// TIA Portal V16 export
// export: Created 2020-03-17T19:45:03.5424607Z, ExportSetting None, DisplayName Totally Integrated Automation Portal, DisplayVersion V16, DisplayName TIA Portal Version Control Interface, DisplayVersion V16, DisplayName TIA Portal Openness, DisplayVersion V16, DisplayName STEP 7 Professional, DisplayVersion V16, DisplayName STEP 7 Safety, DisplayVersion V16, DisplayName WinCC Advanced, DisplayVersion V16
FUNCTION_BLOCK "FB_R134a_GRAPH"   // FB1308, GRAPH
// stored: GraphVersion 2.0, SetENOAutomatically false
   // inherited from GRAPH_BASE
   VAR_INPUT
      OFF_SQ { ExternalAccessible := 'False'; ExternalVisible := 'False'; ExternalWritable := 'False'} : Bool := false;   // Kette ausschalten / Turn sequence off
      INIT_SQ { ExternalAccessible := 'False'; ExternalVisible := 'False'; ExternalWritable := 'False'} : Bool := false;   // Kette in Initialzustand versetzen / Set sequence to initial state
      ACK_EF { ExternalAccessible := 'False'; ExternalVisible := 'False'; ExternalWritable := 'False'} : Bool := false;   // Alle Fehler und Störungen quittieren / Acknowledge all errors and faults
      S_PREV { ExternalAccessible := 'False'; ExternalVisible := 'False'; ExternalWritable := 'False'} : Bool := false;   // Vorherigen Schritt am Parameter S_NO ausgeben / Output previous step in parameter S_NO
      S_NEXT { ExternalAccessible := 'False'; ExternalVisible := 'False'; ExternalWritable := 'False'} : Bool := false;   // Nächsten Schritt am Parameter S_NO anzeigen / Indicate next step in parameter S_NO
      SW_AUTO { ExternalAccessible := 'False'; ExternalVisible := 'False'; ExternalWritable := 'False'} : Bool := false;   // Automatischer Betrieb / Automatic mode
      SW_TAP { ExternalAccessible := 'False'; ExternalVisible := 'False'; ExternalWritable := 'False'} : Bool := false;   // Halbautomatisch/Weiterschalten mit Transition / Semiautomatic/switch with transition
      SW_TOP { ExternalAccessible := 'False'; ExternalVisible := 'False'; ExternalWritable := 'False'} : Bool := false;   // Halbautomatisch/Ignoriere Transition / Semiautomatic/ignore transition
      SW_MAN { ExternalAccessible := 'False'; ExternalVisible := 'False'; ExternalWritable := 'False'} : Bool := false;   // Handbetrieb / Manual mode
      S_SEL { ExternalAccessible := 'False'; ExternalVisible := 'False'; ExternalWritable := 'False'} : Int := 0;   // Schritt auswählen, der an S_NO ausgegeben werden soll / Select step to be output to S_NO
      S_ON { ExternalAccessible := 'False'; ExternalVisible := 'False'; ExternalWritable := 'False'} : Bool := false;   // Schritt aktivieren, der an Parameter S_NO anliegt / Activate step indicated in S_NO
      S_OFF { ExternalAccessible := 'False'; ExternalVisible := 'False'; ExternalWritable := 'False'} : Bool := false;   // Schritt deaktivieren, der an Parameter S_NO anliegt / Deactivate step indicated S_NO
      T_PUSH { ExternalAccessible := 'False'; ExternalVisible := 'False'; ExternalWritable := 'False'} : Bool := false;   // Schaltfreigabe für Transition im halbautomatischen Betrieb / Enable transition to switch in semi automatic mode
   END_VAR
   VAR_OUTPUT
      S_NO { ExternalAccessible := 'False'; ExternalVisible := 'False'; ExternalWritable := 'False'} : Int := 0;   // Schrittnummer / Step number
      S_MORE { ExternalAccessible := 'False'; ExternalVisible := 'False'; ExternalWritable := 'False'} : Bool := false;   // Weitere Schritte sind vorhanden und können in S_NO angezeigt werden. / More steps are available and can be shown in S_NO
      S_ACTIVE { ExternalAccessible := 'False'; ExternalVisible := 'False'; ExternalWritable := 'False'} : Bool := false;   // Schritt, der an Parameter S_NO angezeigt wird, ist aktiv / Step indicated in S_NO is active
      ERR_FLT { ExternalAccessible := 'False'; ExternalVisible := 'False'; ExternalWritable := 'False'} : Bool := false;   // Sammelfehler Interlock oder Supervision / Interlock or supervision group error
      AUTO_ON { ExternalAccessible := 'False'; ExternalVisible := 'False'; ExternalWritable := 'False'} : Bool := false;   // Automatischer Betrieb eingeschaltet / Automatic mode is active
      TAP_ON { ExternalAccessible := 'False'; ExternalVisible := 'False'; ExternalWritable := 'False'} : Bool := false;   // Halbautomatischer Betrieb/Schritt mit Transition eingeschaltet / Semiautomatic mode/step with transition enabled
      TOP_ON { ExternalAccessible := 'False'; ExternalVisible := 'False'; ExternalWritable := 'False'} : Bool := false;   // Halbautomatischer Betrieb/Ignoriere Transition eingeschaltet / Semiautomatic mode/ignore transition enabled
      MAN_ON { ExternalAccessible := 'False'; ExternalVisible := 'False'; ExternalWritable := 'False'} : Bool := false;   // Handbetrieb eingeschaltet / Manual mode is active
   END_VAR
BEGIN
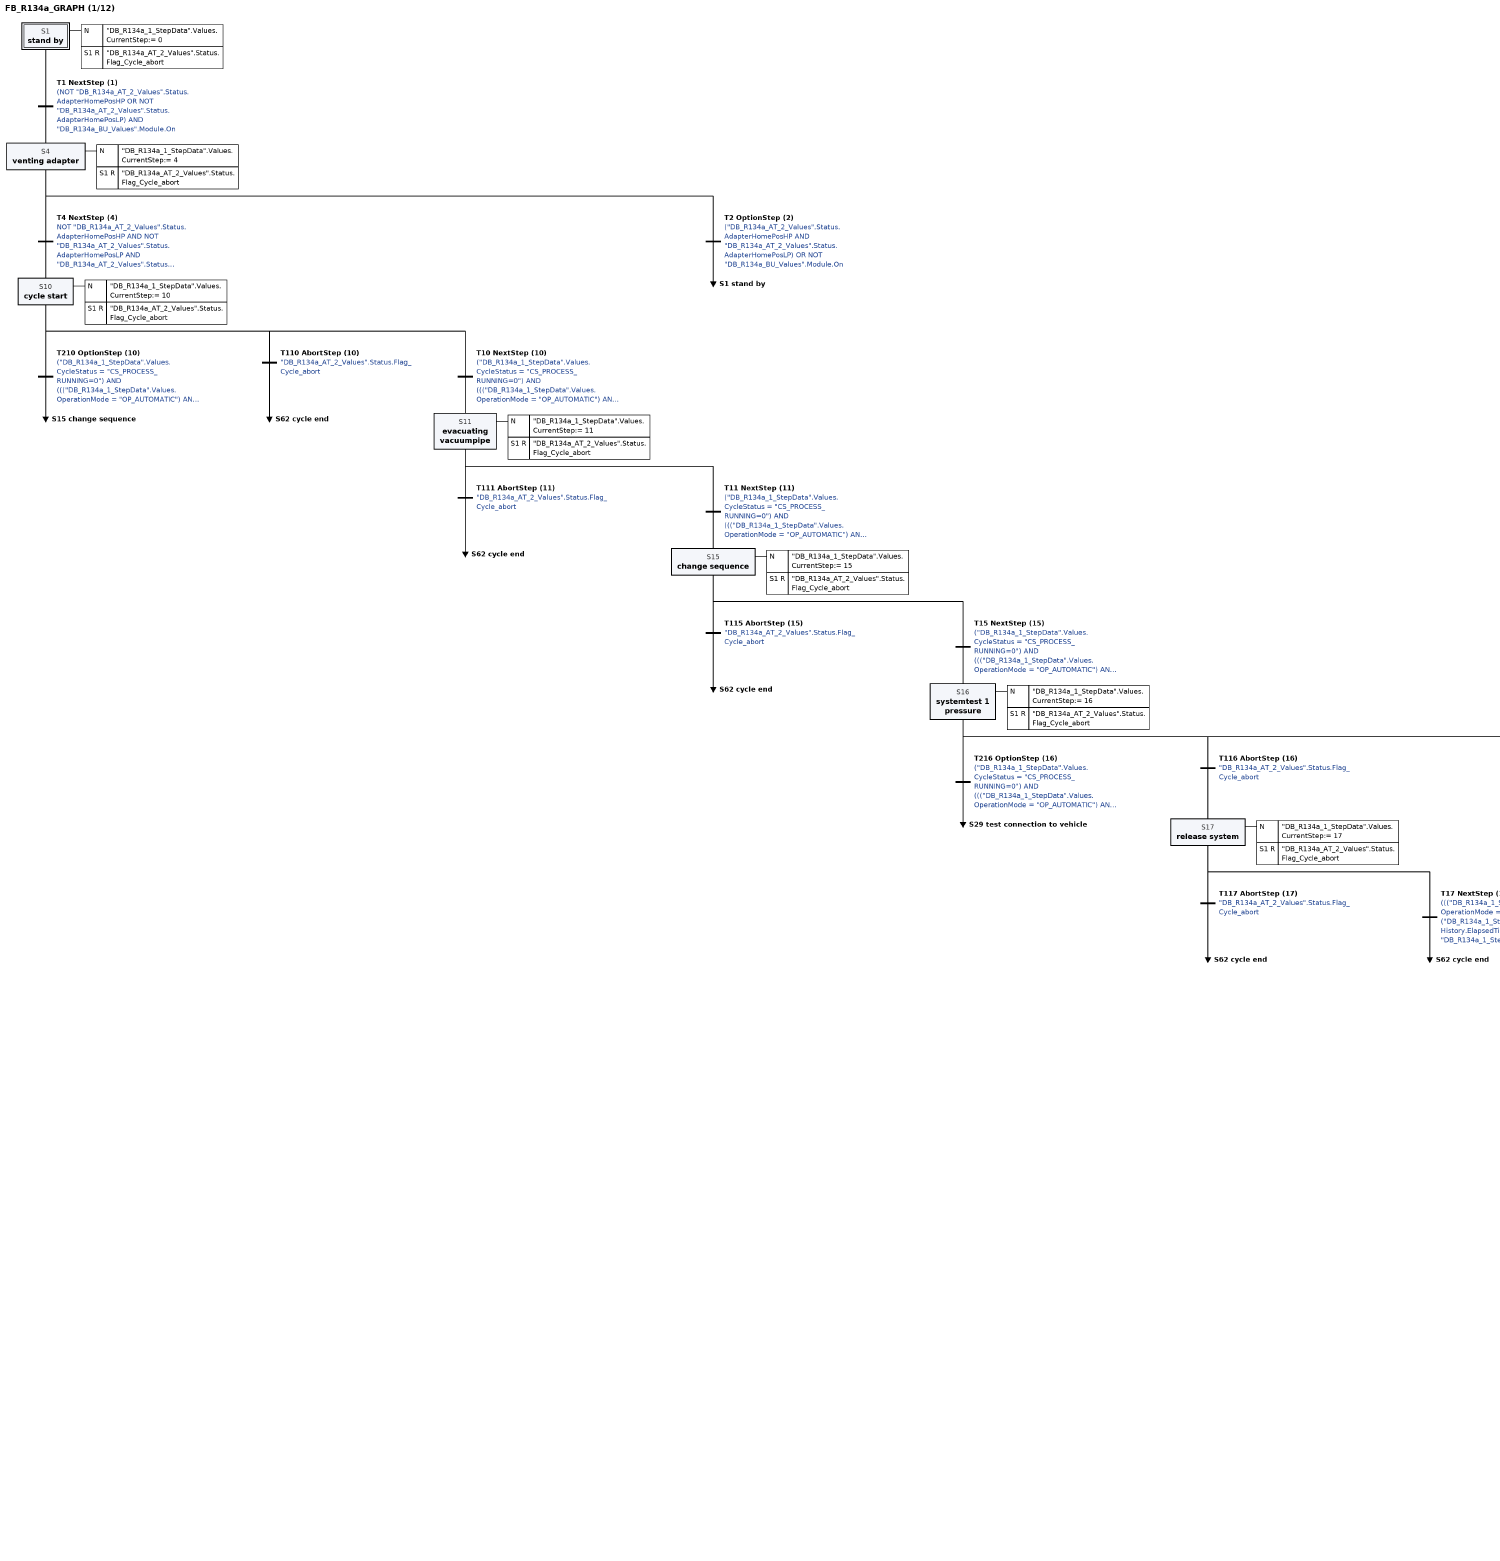
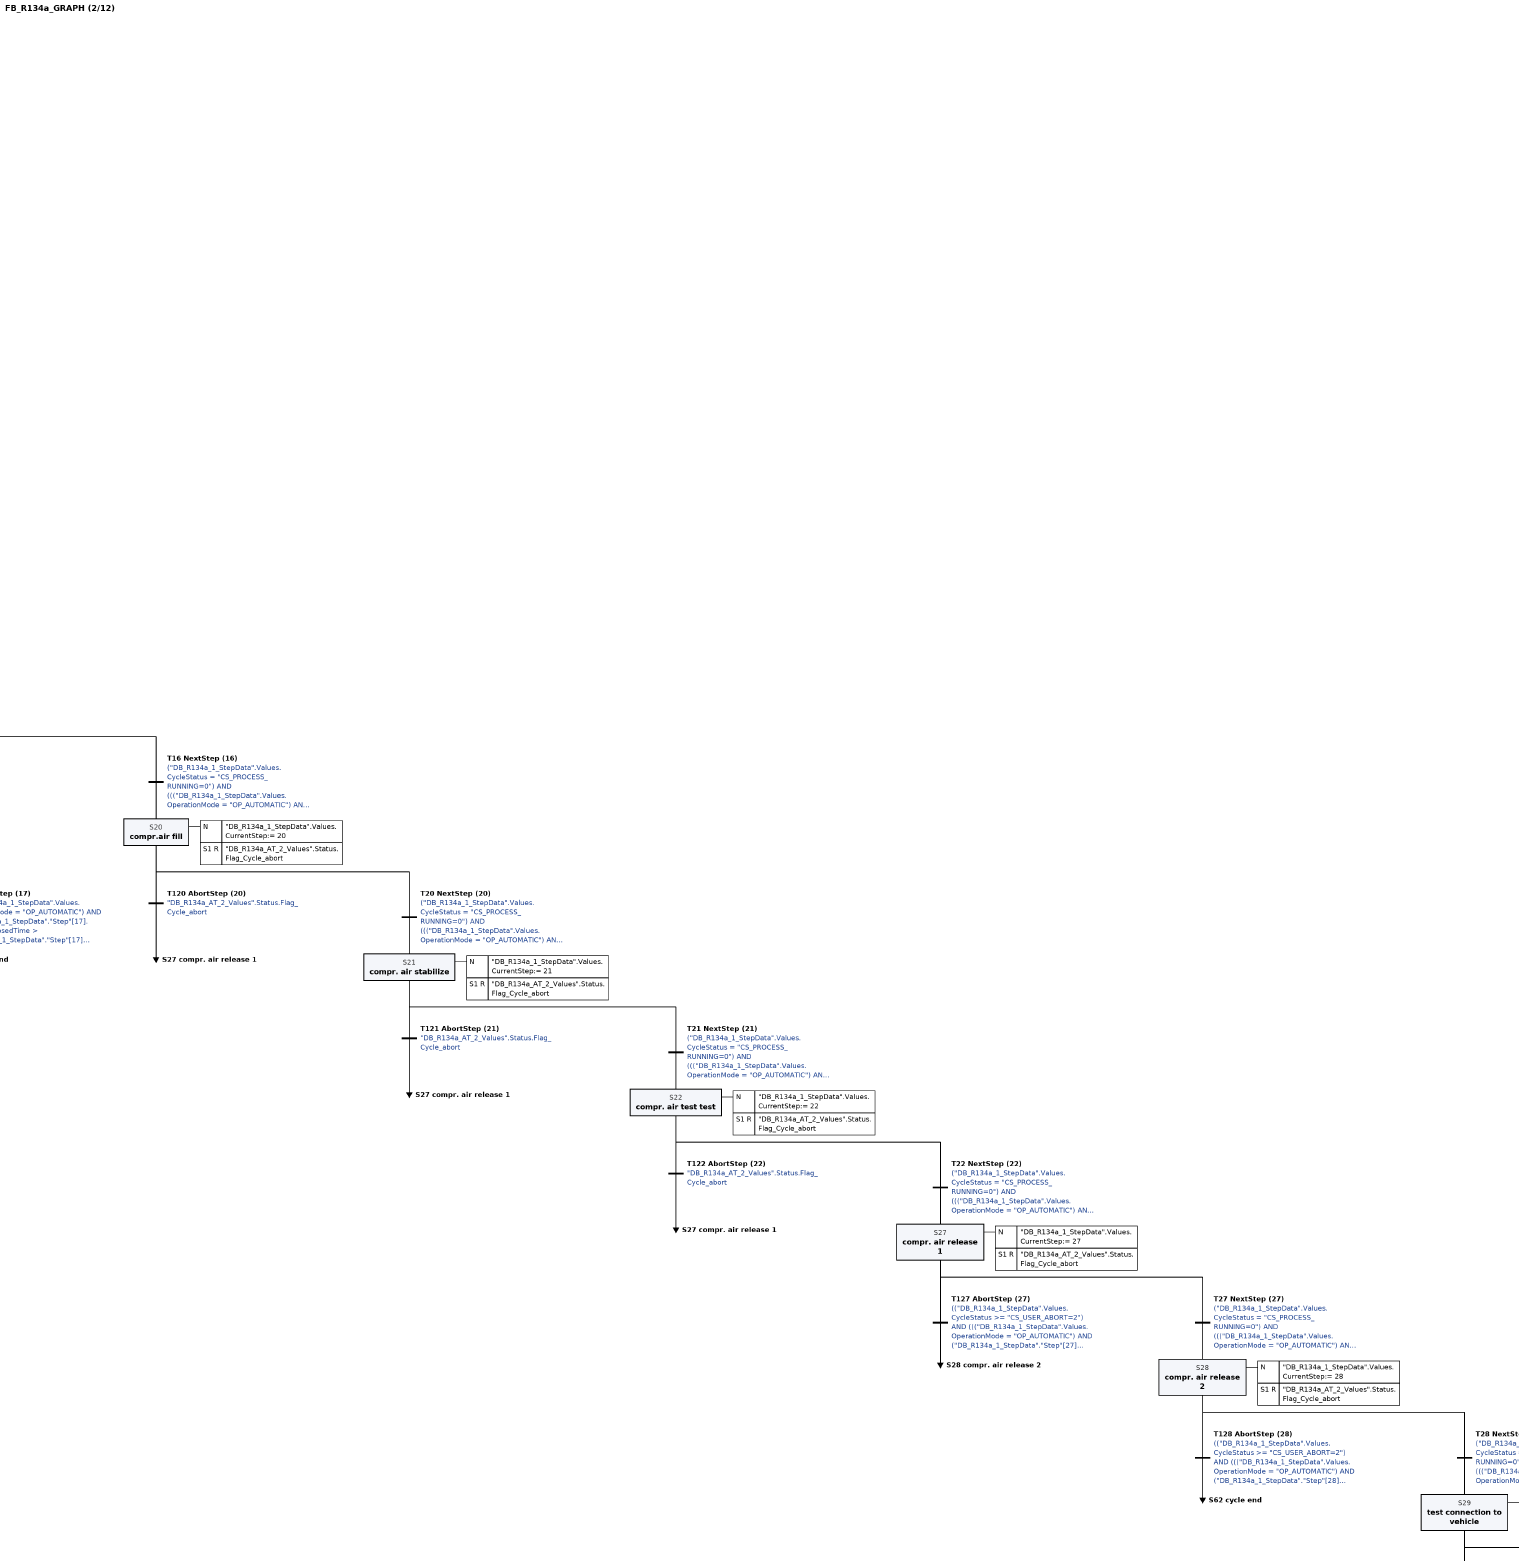
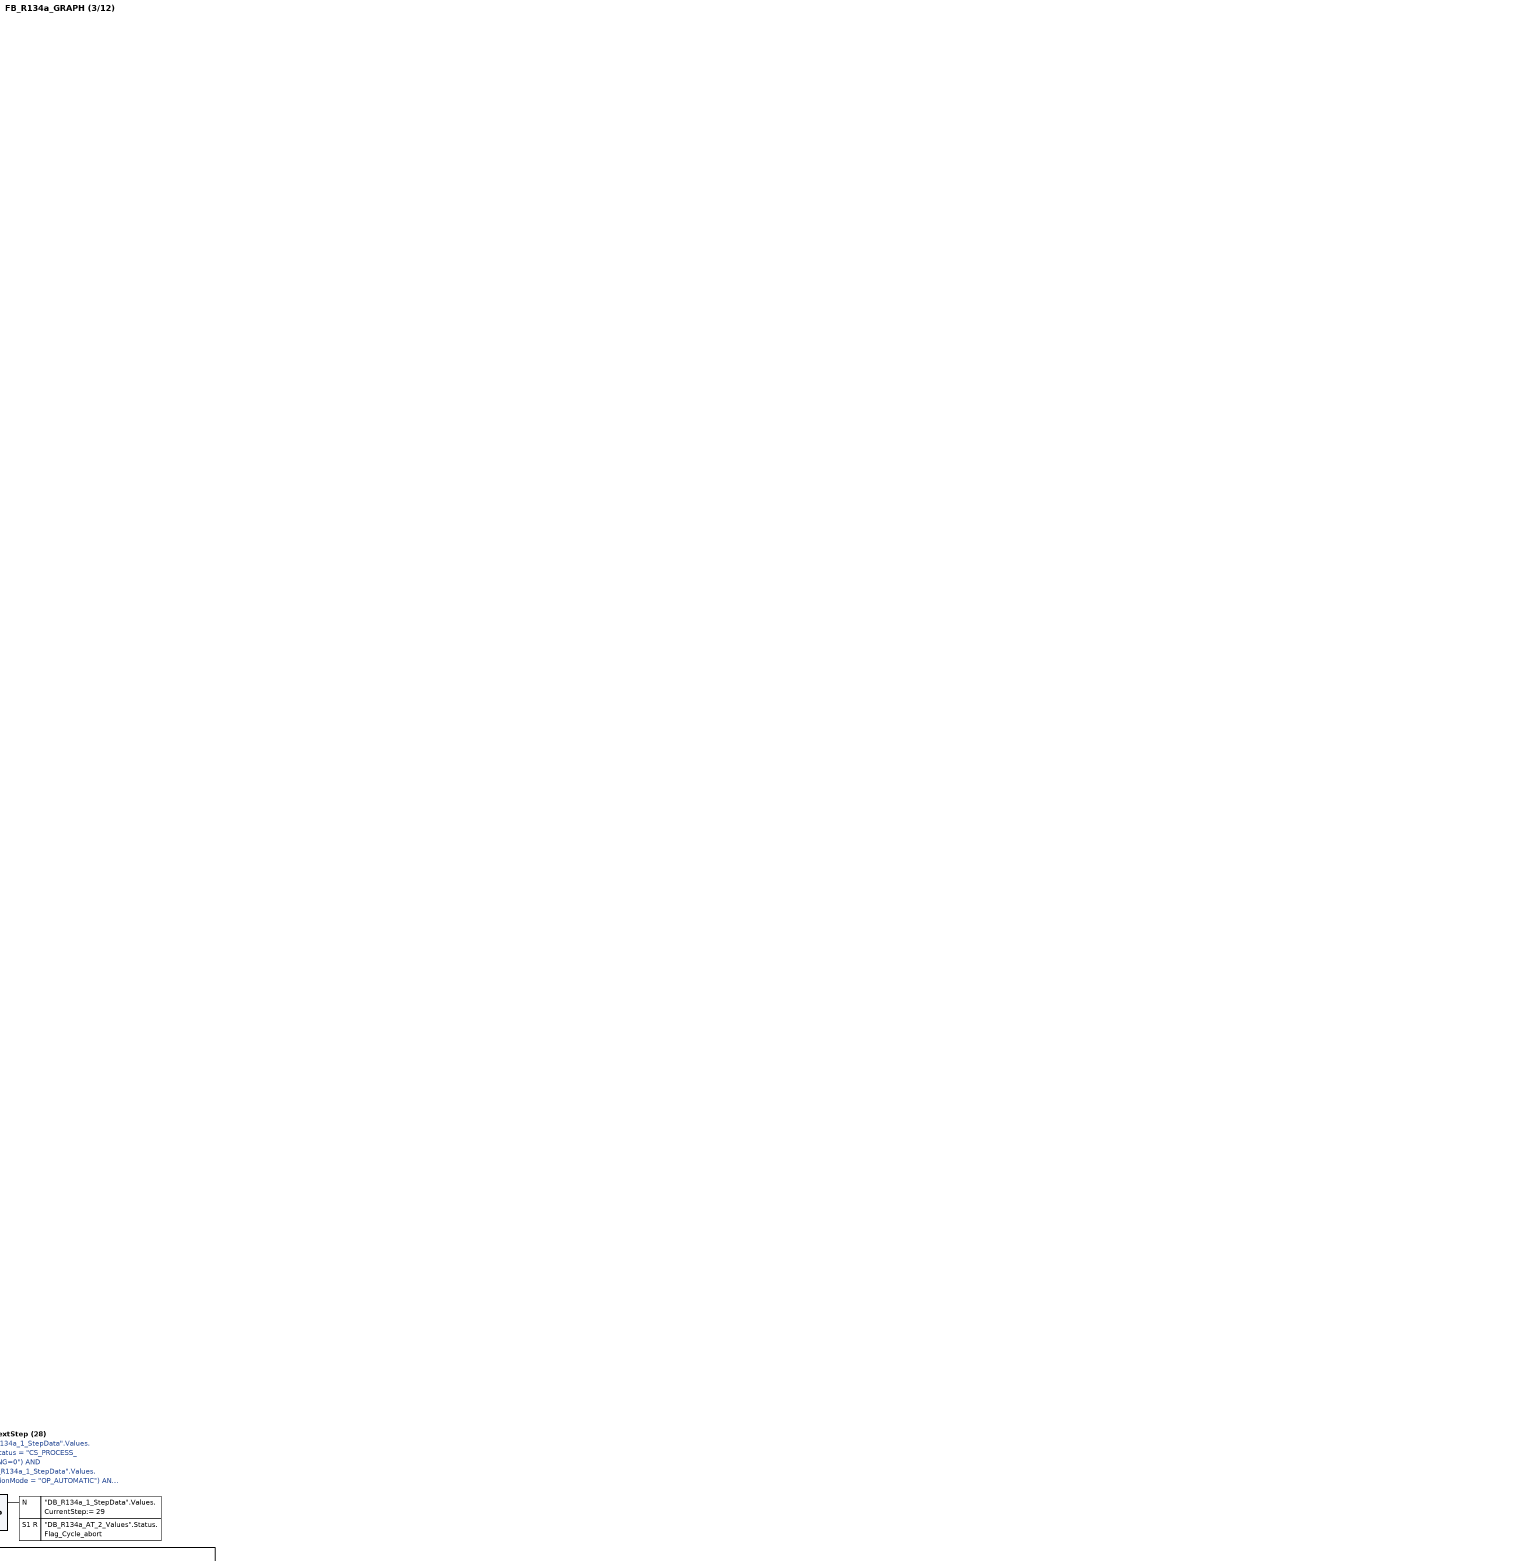
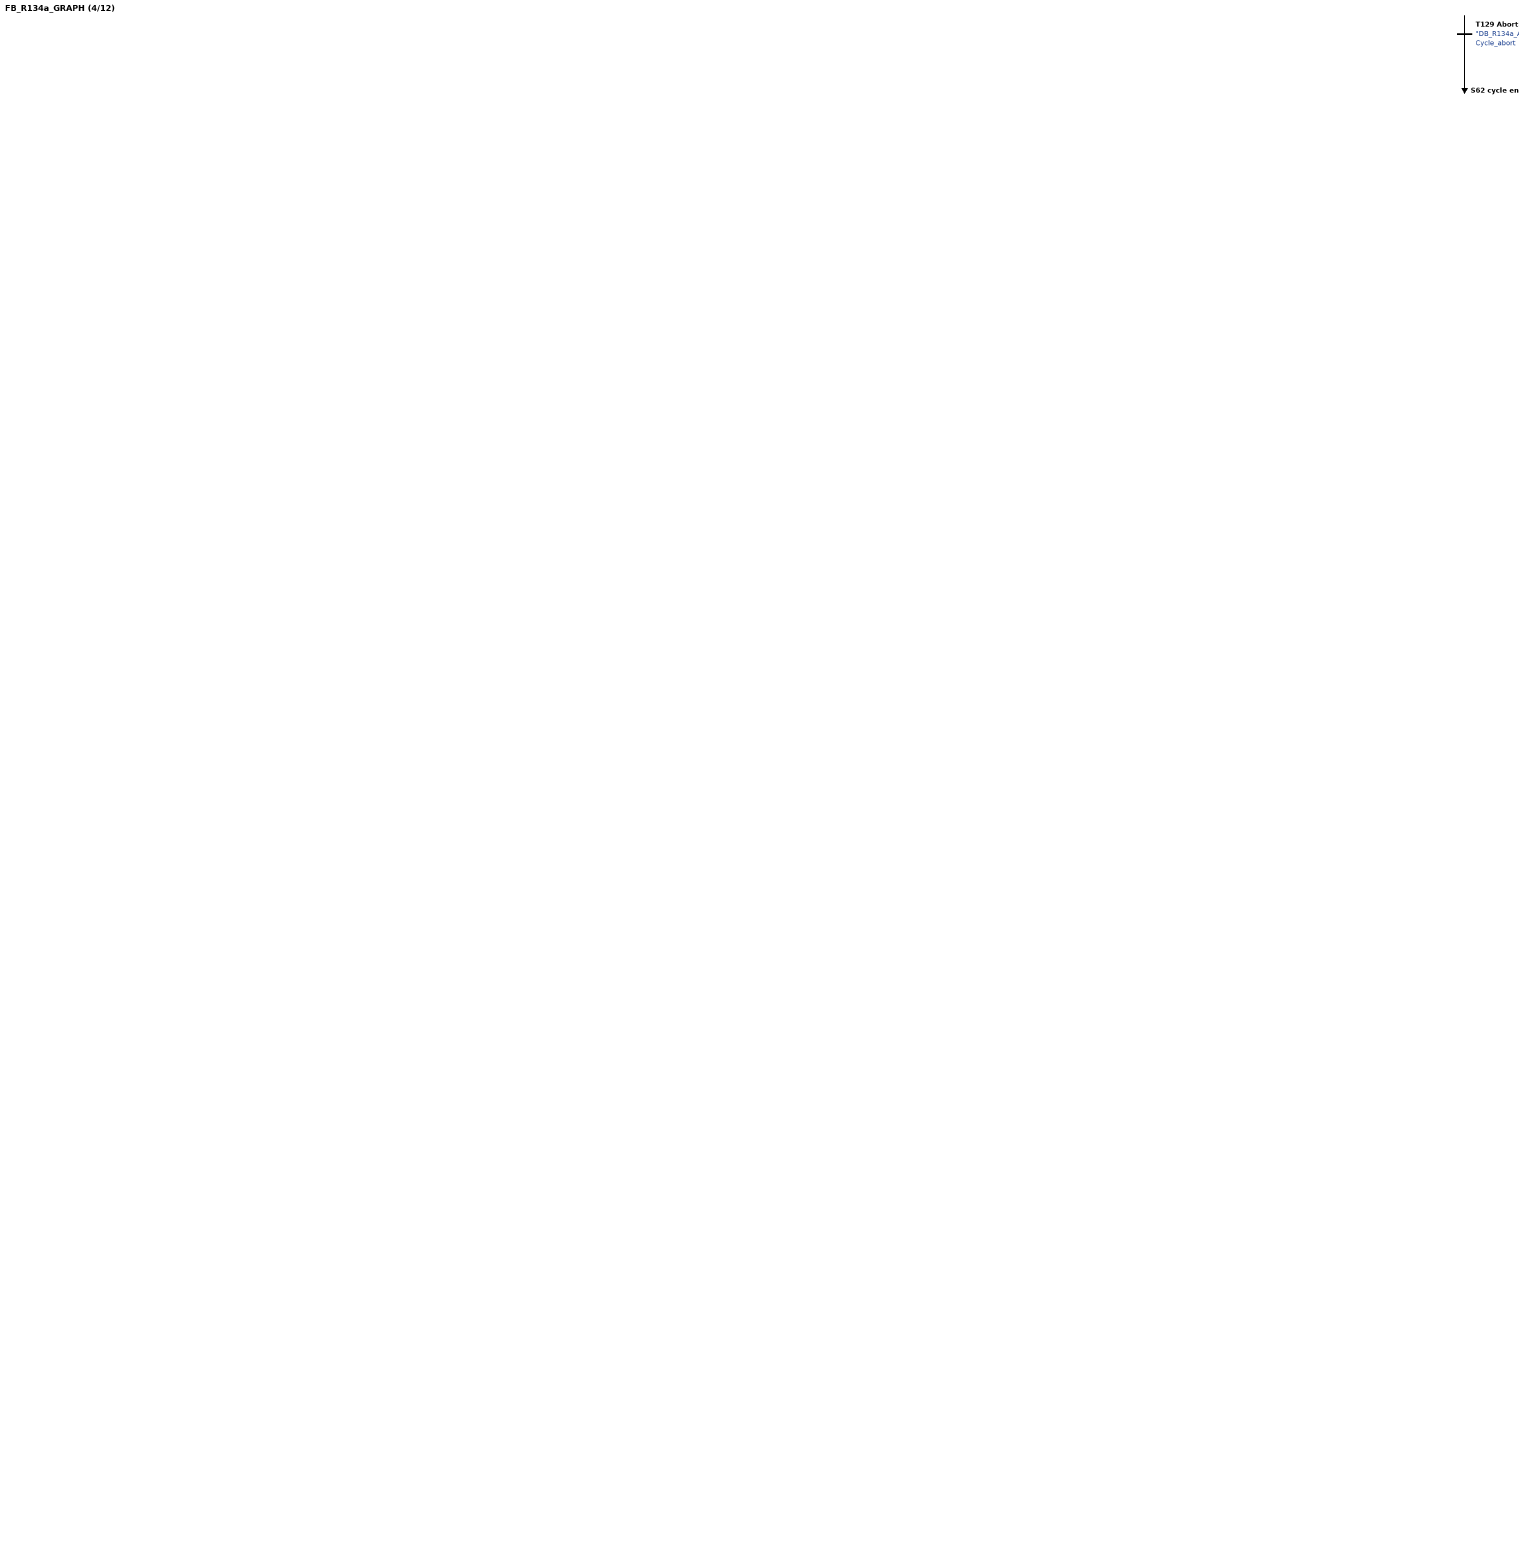
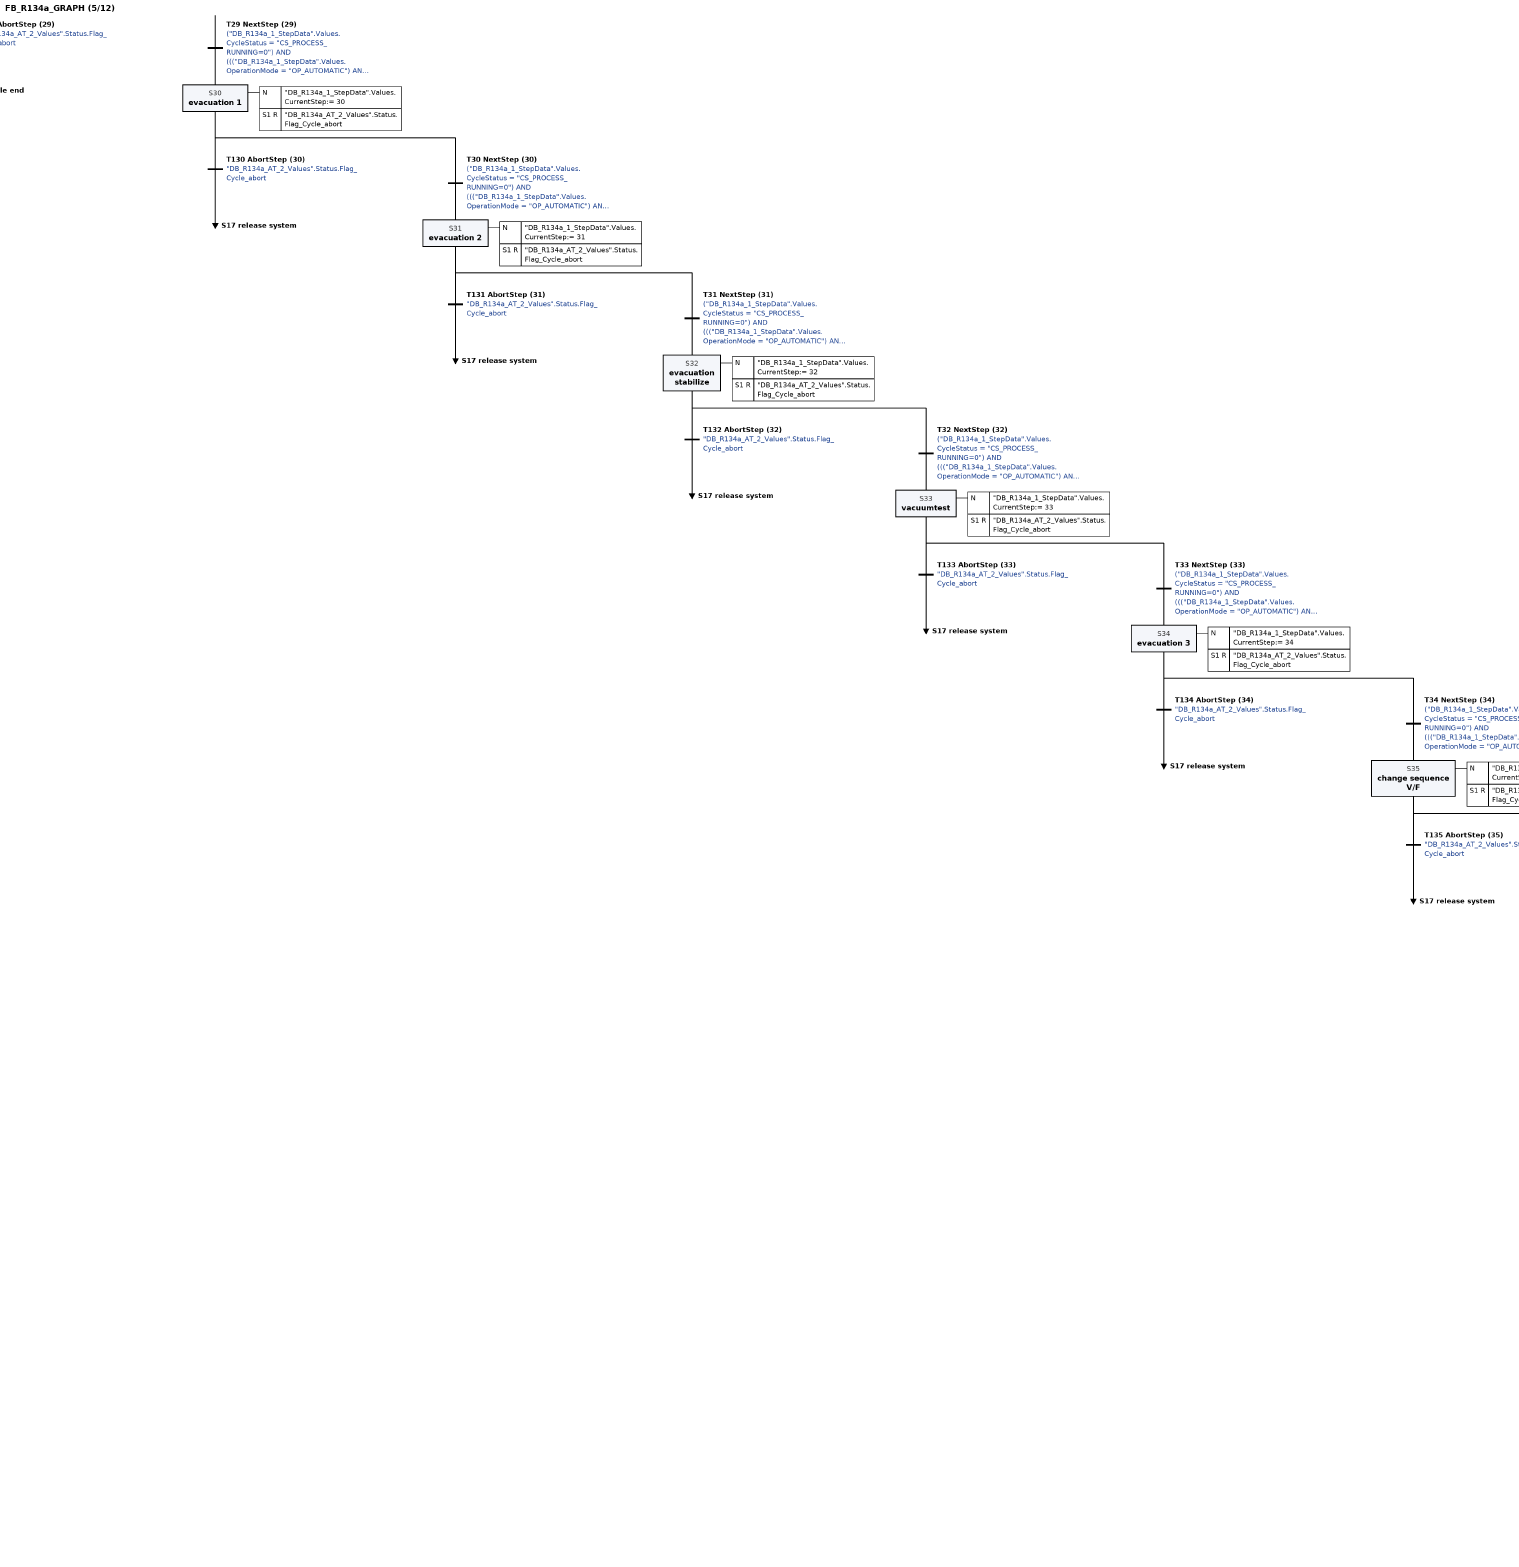
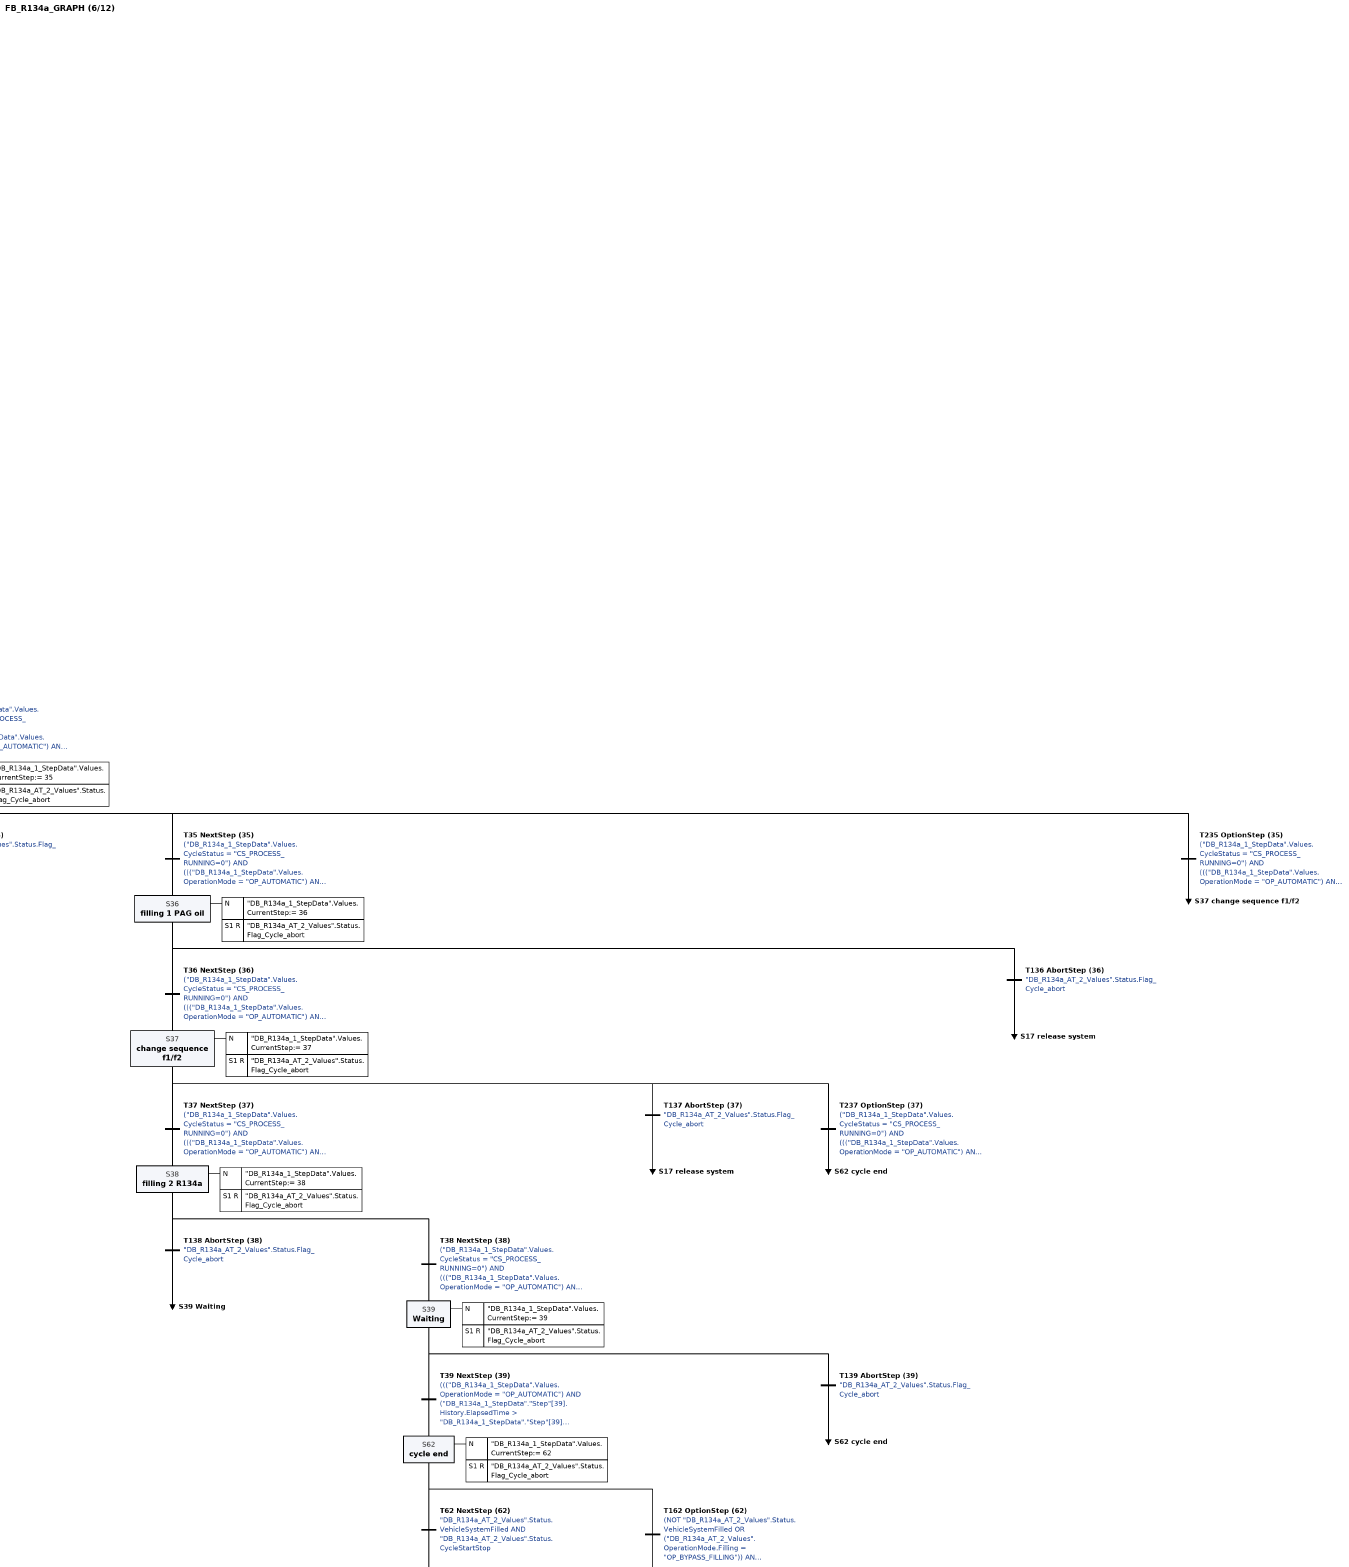
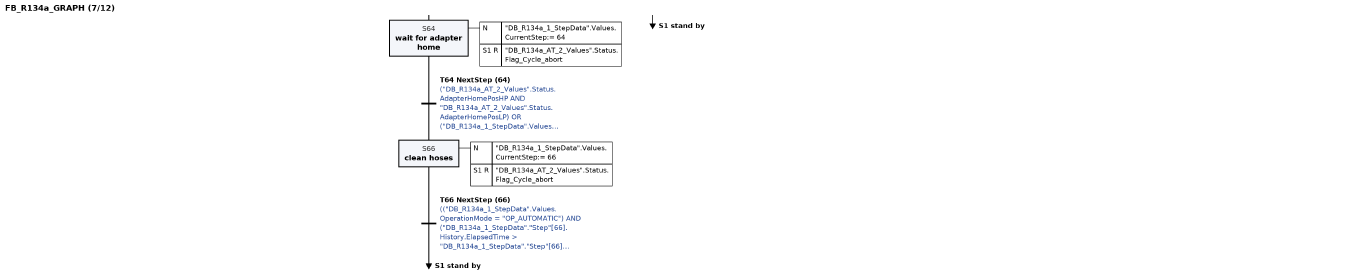
   // sequencer 1
   STEP "release system":   // S17, max time T#10S, warning time T#7S
              N    "DB_R134a_1_StepData".Values.CurrentStep:= 17
          S1  R    "DB_R134a_AT_2_Values".Status.Flag_Cycle_abort
   END_STEP
   TRANSITION "AbortStep (17)" FROM "release system" TO "cycle end"   // T117, jump
      := "DB_R134a_AT_2_Values".Status.Flag_Cycle_abort;
   END_TRANSITION
   TRANSITION "NextStep (17)" FROM "release system" TO "cycle end"   // T17, jump
      := ((("DB_R134a_1_StepData".Values.OperationMode = "OP_AUTOMATIC") AND ("DB_R134a_1_StepData"."Step"[17].History.ElapsedTime > "DB_R134a_1_StepData"."Step"[17].WaitingTime)) OR ("DB_R134a_1_StepData".Values.SingleStep AND ("DB_R134a_1_StepData".Values.OperationMode = "OP_SingleStep"))) AND NOT "DB_R134a_AT_2_Values".Status.Flag_Cycle_abort;
   END_TRANSITION
   STEP "clean hoses":   // S66, max time T#10S, warning time T#7S
              N    "DB_R134a_1_StepData".Values.CurrentStep:= 66
          S1  R    "DB_R134a_AT_2_Values".Status.Flag_Cycle_abort
   END_STEP
   TRANSITION "NextStep (66)" FROM "clean hoses" TO "stand by"   // T66, jump
      := (("DB_R134a_1_StepData".Values.OperationMode = "OP_AUTOMATIC") AND ("DB_R134a_1_StepData"."Step"[66].History.ElapsedTime > "DB_R134a_1_StepData"."Step"[66].WaitingTime)) OR ("DB_R134a_1_StepData".Values.SingleStep AND ("DB_R134a_1_StepData".Values.OperationMode = "OP_SingleStep"));
   END_TRANSITION
   STEP "wait for adapter home":   // S64, max time T#10S, warning time T#7S
              N    "DB_R134a_1_StepData".Values.CurrentStep:= 64
          S1  R    "DB_R134a_AT_2_Values".Status.Flag_Cycle_abort
   END_STEP
   TRANSITION "NextStep (64)" FROM "wait for adapter home" TO "clean hoses"   // T64
      := ("DB_R134a_AT_2_Values".Status.AdapterHomePosHP AND "DB_R134a_AT_2_Values".Status.AdapterHomePosLP) OR ("DB_R134a_1_StepData".Values.SingleStep AND ("DB_R134a_1_StepData".Values.OperationMode = "OP_SingleStep"));
   END_TRANSITION
   STEP "cycle end":   // S62, max time T#10S, warning time T#7S
              N    "DB_R134a_1_StepData".Values.CurrentStep:= 62
          S1  R    "DB_R134a_AT_2_Values".Status.Flag_Cycle_abort
   END_STEP
   TRANSITION "NextStep (62)" FROM "cycle end" TO "wait for adapter home"   // T62
      := "DB_R134a_AT_2_Values".Status.VehicleSystemFilled AND "DB_R134a_AT_2_Values".Status.CycleStartStop;
   END_TRANSITION
   TRANSITION "OptionStep (62)" FROM "cycle end" TO "stand by"   // T162, jump
      := (NOT "DB_R134a_AT_2_Values".Status.VehicleSystemFilled OR ("DB_R134a_AT_2_Values".OperationMode.Filling = "OP_BYPASS_FILLING")) AND "DB_R134a_AT_2_Values".Status.CycleStartStop;
   END_TRANSITION
   STEP Waiting:   // S39, max time T#10S, warning time T#7S
              N    "DB_R134a_1_StepData".Values.CurrentStep:= 39
          S1  R    "DB_R134a_AT_2_Values".Status.Flag_Cycle_abort
   END_STEP
   TRANSITION "NextStep (39)" FROM Waiting TO "cycle end"   // T39
      := ((("DB_R134a_1_StepData".Values.OperationMode = "OP_AUTOMATIC") AND ("DB_R134a_1_StepData"."Step"[39].History.ElapsedTime > "DB_R134a_1_StepData"."Step"[39].WaitingTime)) OR ("DB_R134a_1_StepData".Values.SingleStep AND ("DB_R134a_1_StepData".Values.OperationMode = "OP_SingleStep"))) AND NOT "DB_R134a_AT_2_Values".Status.Flag_Cycle_abort;
   END_TRANSITION
   TRANSITION "AbortStep (39)" FROM Waiting TO "cycle end"   // T139, jump
      := "DB_R134a_AT_2_Values".Status.Flag_Cycle_abort;
   END_TRANSITION
   STEP "filling 2 R134a":   // S38, max time T#10S, warning time T#7S
      supervision V := ("DB_R134a_1_StepData".Values.OperationMode <> "OP_SingleStep") AND (#"filling 2 R134a".U > "DB_R134a_1_StepData"."Step"[38].MonitoringTime) AND ("DB_R134a_1_StepData".Values.CycleStatus = "CS_PROCESS_RUNNING=0");
              N    "DB_R134a_1_StepData".Values.CurrentStep:= 38
          S1  R    "DB_R134a_AT_2_Values".Status.Flag_Cycle_abort
   END_STEP
   TRANSITION "AbortStep (38)" FROM "filling 2 R134a" TO Waiting   // T138, jump
      := "DB_R134a_AT_2_Values".Status.Flag_Cycle_abort;
   END_TRANSITION
   TRANSITION "NextStep (38)" FROM "filling 2 R134a" TO Waiting   // T38
      := ("DB_R134a_1_StepData".Values.CycleStatus = "CS_PROCESS_RUNNING=0") AND ((("DB_R134a_1_StepData".Values.OperationMode = "OP_AUTOMATIC") AND ("DB_R134a_1_StepData"."Step"[38].History.ElapsedTime > "DB_R134a_1_StepData"."Step"[38].WaitingTime) AND "DB_R134a_BU_Values".Flowmeter.Output.VolumeDone) OR ("DB_R134a_1_StepData".Values.SingleStep AND ("DB_R134a_1_StepData".Values.OperationMode = "OP_SingleStep"))) AND NOT "DB_R134a_AT_2_Values".Status.Flag_Cycle_abort;
   END_TRANSITION
   STEP "change sequence V/F":   // S35, max time T#10S, warning time T#7S
              N    "DB_R134a_1_StepData".Values.CurrentStep:= 35
          S1  R    "DB_R134a_AT_2_Values".Status.Flag_Cycle_abort
   END_STEP
   TRANSITION "AbortStep (35)" FROM "change sequence V/F" TO "release system"   // T135, jump
      := "DB_R134a_AT_2_Values".Status.Flag_Cycle_abort;
   END_TRANSITION
   TRANSITION "NextStep (35)" FROM "change sequence V/F" TO "filling 1 PAG oil"   // T35
      := ("DB_R134a_1_StepData".Values.CycleStatus = "CS_PROCESS_RUNNING=0") AND ((("DB_R134a_1_StepData".Values.OperationMode = "OP_AUTOMATIC") AND ("DB_R134a_1_StepData"."Step"[35].History.ElapsedTime > "DB_R134a_1_StepData"."Step"[35].WaitingTime)) OR ("DB_R134a_1_StepData".Values.SingleStep AND ("DB_R134a_1_StepData".Values.OperationMode = "OP_SingleStep"))) AND ("DB_R134a_AT_2_Values".OperationMode.FillingPAG = "OP_WITH_PAG") AND NOT "DB_R134a_AT_2_Values".Status.Flag_Cycle_abort;
   END_TRANSITION
   TRANSITION "OptionStep (35)" FROM "change sequence V/F" TO "change sequence f1/f2"   // T235, jump
      := ("DB_R134a_1_StepData".Values.CycleStatus = "CS_PROCESS_RUNNING=0") AND ((("DB_R134a_1_StepData".Values.OperationMode = "OP_AUTOMATIC") AND ("DB_R134a_1_StepData"."Step"[35].History.ElapsedTime > "DB_R134a_1_StepData"."Step"[35].WaitingTime)) OR ("DB_R134a_1_StepData".Values.SingleStep AND ("DB_R134a_1_StepData".Values.OperationMode = "OP_SingleStep"))) AND ("DB_R134a_AT_2_Values".OperationMode.FillingPAG = "OP_BYPASS_FILLING_PAG") AND NOT "DB_R134a_AT_2_Values".Status.Flag_Cycle_abort;
   END_TRANSITION
   STEP "evacuation 3":   // S34, max time T#10S, warning time T#7S
      supervision V := ("DB_R134a_1_StepData".Values.OperationMode <> "OP_SingleStep") AND (#"evacuation 3".U > "DB_R134a_1_StepData"."Step"[34].MonitoringTime) AND ("DB_R134a_1_StepData".Values.CycleStatus = "CS_PROCESS_RUNNING=0");
              N    "DB_R134a_1_StepData".Values.CurrentStep:= 34
          S1  R    "DB_R134a_AT_2_Values".Status.Flag_Cycle_abort
   END_STEP
   TRANSITION "AbortStep (34)" FROM "evacuation 3" TO "release system"   // T134, jump
      := "DB_R134a_AT_2_Values".Status.Flag_Cycle_abort;
   END_TRANSITION
   TRANSITION "NextStep (34)" FROM "evacuation 3" TO "change sequence V/F"   // T34
      := ("DB_R134a_1_StepData".Values.CycleStatus = "CS_PROCESS_RUNNING=0") AND ((("DB_R134a_1_StepData".Values.OperationMode = "OP_AUTOMATIC") AND ("DB_R134a_1_StepData"."Step"[34].History.ElapsedTime > "DB_R134a_1_StepData"."Step"[34].WaitingTime) AND ("DB_R134a_1_StepData"."Step"[34].History.Values[1] <= "DB_R134a_1_StepData"."Step"[34].Setpoint[1])) OR ("DB_R134a_1_StepData".Values.SingleStep AND ("DB_R134a_1_StepData".Values.OperationMode = "OP_SingleStep"))) AND NOT "DB_R134a_AT_2_Values".Status.Flag_Cycle_abort;
   END_TRANSITION
   STEP vacuumtest:   // S33, max time T#10S, warning time T#7S
      supervision V := ("DB_R134a_1_StepData".Values.OperationMode <> "OP_SingleStep") AND (#vacuumtest.U > "DB_R134a_1_StepData"."Step"[33].MonitoringTime) AND ("DB_R134a_1_StepData".Values.CycleStatus = "CS_PROCESS_RUNNING=0");
              N    "DB_R134a_1_StepData".Values.CurrentStep:= 33
          S1  R    "DB_R134a_AT_2_Values".Status.Flag_Cycle_abort
   END_STEP
   TRANSITION "AbortStep (33)" FROM vacuumtest TO "release system"   // T133, jump
      := "DB_R134a_AT_2_Values".Status.Flag_Cycle_abort;
   END_TRANSITION
   TRANSITION "NextStep (33)" FROM vacuumtest TO "evacuation 3"   // T33
      := ("DB_R134a_1_StepData".Values.CycleStatus = "CS_PROCESS_RUNNING=0") AND ((("DB_R134a_1_StepData".Values.OperationMode = "OP_AUTOMATIC") AND ("DB_R134a_1_StepData"."Step"[33].History.ElapsedTime > "DB_R134a_1_StepData"."Step"[33].WaitingTime) AND ("DB_R134a_1_StepData"."Step"[33].History.Values[1] <= "DB_R134a_1_StepData"."Step"[33].Setpoint[1]) AND ("DB_R134a_1_StepData"."Step"[33].History.Values[2] <= "DB_R134a_1_StepData"."Step"[33].Setpoint[2])) OR ("DB_R134a_1_StepData".Values.SingleStep AND ("DB_R134a_1_StepData".Values.OperationMode = "OP_SingleStep"))) AND NOT "DB_R134a_AT_2_Values".Status.Flag_Cycle_abort;
   END_TRANSITION
   STEP "evacuation stabilize":   // S32, max time T#10S, warning time T#7S
              N    "DB_R134a_1_StepData".Values.CurrentStep:= 32
          S1  R    "DB_R134a_AT_2_Values".Status.Flag_Cycle_abort
   END_STEP
   TRANSITION "AbortStep (32)" FROM "evacuation stabilize" TO "release system"   // T132, jump
      := "DB_R134a_AT_2_Values".Status.Flag_Cycle_abort;
   END_TRANSITION
   TRANSITION "NextStep (32)" FROM "evacuation stabilize" TO vacuumtest   // T32
      := ("DB_R134a_1_StepData".Values.CycleStatus = "CS_PROCESS_RUNNING=0") AND ((("DB_R134a_1_StepData".Values.OperationMode = "OP_AUTOMATIC") AND ("DB_R134a_1_StepData"."Step"[32].History.ElapsedTime > "DB_R134a_1_StepData"."Step"[32].WaitingTime)) OR ("DB_R134a_1_StepData".Values.SingleStep AND ("DB_R134a_1_StepData".Values.OperationMode = "OP_SingleStep"))) AND NOT "DB_R134a_AT_2_Values".Status.Flag_Cycle_abort;
   END_TRANSITION
   STEP "evacuation 2":   // S31, max time T#10S, warning time T#7S
      supervision V := ("DB_R134a_1_StepData".Values.OperationMode <> "OP_SingleStep") AND (#"evacuation 2".U > "DB_R134a_1_StepData"."Step"[31].MonitoringTime) AND ("DB_R134a_1_StepData".Values.CycleStatus = "CS_PROCESS_RUNNING=0");
              N    "DB_R134a_1_StepData".Values.CurrentStep:= 31
          S1  R    "DB_R134a_AT_2_Values".Status.Flag_Cycle_abort
   END_STEP
   TRANSITION "AbortStep (31)" FROM "evacuation 2" TO "release system"   // T131, jump
      := "DB_R134a_AT_2_Values".Status.Flag_Cycle_abort;
   END_TRANSITION
   TRANSITION "NextStep (31)" FROM "evacuation 2" TO "evacuation stabilize"   // T31
      := ("DB_R134a_1_StepData".Values.CycleStatus = "CS_PROCESS_RUNNING=0") AND ((("DB_R134a_1_StepData".Values.OperationMode = "OP_AUTOMATIC") AND ("DB_R134a_1_StepData"."Step"[31].History.ElapsedTime > "DB_R134a_1_StepData"."Step"[31].WaitingTime) AND ("DB_R134a_1_StepData"."Step"[31].History.Values[1] <= "DB_R134a_1_StepData"."Step"[31].Setpoint[1])) OR ("DB_R134a_1_StepData".Values.SingleStep AND ("DB_R134a_1_StepData".Values.OperationMode = "OP_SingleStep"))) AND NOT "DB_R134a_AT_2_Values".Status.Flag_Cycle_abort;
   END_TRANSITION
   STEP "evacuation 1":   // S30, max time T#10S, warning time T#7S
      supervision V := ("DB_R134a_1_StepData".Values.OperationMode <> "OP_SingleStep") AND (#"evacuation 1".U > "DB_R134a_1_StepData"."Step"[30].MonitoringTime) AND ("DB_R134a_1_StepData".Values.CycleStatus = "CS_PROCESS_RUNNING=0");
              N    "DB_R134a_1_StepData".Values.CurrentStep:= 30
          S1  R    "DB_R134a_AT_2_Values".Status.Flag_Cycle_abort
   END_STEP
   TRANSITION "AbortStep (30)" FROM "evacuation 1" TO "release system"   // T130, jump
      := "DB_R134a_AT_2_Values".Status.Flag_Cycle_abort;
   END_TRANSITION
   TRANSITION "NextStep (30)" FROM "evacuation 1" TO "evacuation 2"   // T30
      := ("DB_R134a_1_StepData".Values.CycleStatus = "CS_PROCESS_RUNNING=0") AND ((("DB_R134a_1_StepData".Values.OperationMode = "OP_AUTOMATIC") AND ("DB_R134a_1_StepData"."Step"[30].History.ElapsedTime > "DB_R134a_1_StepData"."Step"[30].WaitingTime) AND ("DB_R134a_1_StepData"."Step"[30].History.Values[1] <= "DB_R134a_1_StepData"."Step"[30].Setpoint[1])) OR ("DB_R134a_1_StepData".Values.SingleStep AND ("DB_R134a_1_StepData".Values.OperationMode = "OP_SingleStep"))) AND NOT "DB_R134a_AT_2_Values".Status.Flag_Cycle_abort;
   END_TRANSITION
   STEP "test connection to vehicle":   // S29, max time T#10S, warning time T#7S
      supervision V := ("DB_R134a_1_StepData".Values.OperationMode <> "OP_SingleStep") AND (#"test connection to vehicle".U > "DB_R134a_1_StepData"."Step"[29].MonitoringTime) AND ("DB_R134a_1_StepData".Values.CycleStatus = "CS_PROCESS_RUNNING=0");
              N    "DB_R134a_1_StepData".Values.CurrentStep:= 29
          S1  R    "DB_R134a_AT_2_Values".Status.Flag_Cycle_abort
   END_STEP
   TRANSITION "AbortStep (29)" FROM "test connection to vehicle" TO "cycle end"   // T129, jump
      := "DB_R134a_AT_2_Values".Status.Flag_Cycle_abort;
   END_TRANSITION
   TRANSITION "NextStep (29)" FROM "test connection to vehicle" TO "evacuation 1"   // T29
      := ("DB_R134a_1_StepData".Values.CycleStatus = "CS_PROCESS_RUNNING=0") AND ((("DB_R134a_1_StepData".Values.OperationMode = "OP_AUTOMATIC") AND ("DB_R134a_1_StepData"."Step"[29].History.ElapsedTime > "DB_R134a_1_StepData"."Step"[29].WaitingTime) AND ("DB_R134a_1_StepData"."Step"[29].History.Values[1] >= "DB_R134a_1_StepData"."Step"[29].Setpoint[1])) OR ("DB_R134a_1_StepData".Values.SingleStep AND ("DB_R134a_1_StepData".Values.OperationMode = "OP_SingleStep"))) AND NOT "DB_R134a_AT_2_Values".Status.Flag_Cycle_abort;
   END_TRANSITION
   STEP "compr. air release 2":   // S28, max time T#10S, warning time T#7S
      supervision V := ("DB_R134a_1_StepData".Values.OperationMode <> "OP_SingleStep") AND (#"compr. air release 2".U > "DB_R134a_1_StepData"."Step"[28].MonitoringTime) AND ("DB_R134a_1_StepData".Values.CycleStatus = "CS_PROCESS_RUNNING=0");
              N    "DB_R134a_1_StepData".Values.CurrentStep:= 28
          S1  R    "DB_R134a_AT_2_Values".Status.Flag_Cycle_abort
   END_STEP
   TRANSITION "AbortStep (28)" FROM "compr. air release 2" TO "cycle end"   // T128, jump
      := (("DB_R134a_1_StepData".Values.CycleStatus >= "CS_USER_ABORT=2") AND ((("DB_R134a_1_StepData".Values.OperationMode = "OP_AUTOMATIC") AND ("DB_R134a_1_StepData"."Step"[28].History.ElapsedTime > "DB_R134a_1_StepData"."Step"[28].WaitingTime)) OR ("DB_R134a_1_StepData".Values.SingleStep AND ("DB_R134a_1_StepData".Values.OperationMode = "OP_SingleStep"))) AND NOT "DB_R134a_AT_2_Values".Status.Flag_Cycle_abort) OR "DB_R134a_AT_2_Values".Status.Flag_Cycle_abort;
   END_TRANSITION
   TRANSITION "NextStep (28)" FROM "compr. air release 2" TO "test connection to vehicle"   // T28
      := ("DB_R134a_1_StepData".Values.CycleStatus = "CS_PROCESS_RUNNING=0") AND ((("DB_R134a_1_StepData".Values.OperationMode = "OP_AUTOMATIC") AND ("DB_R134a_1_StepData"."Step"[28].History.ElapsedTime > "DB_R134a_1_StepData"."Step"[28].WaitingTime) AND ("DB_R134a_1_StepData"."Step"[28].History.Values[5] <= "DB_R134a_1_StepData"."Step"[28].Setpoint[5])) OR ("DB_R134a_1_StepData".Values.SingleStep AND ("DB_R134a_1_StepData".Values.OperationMode = "OP_SingleStep"))) AND NOT "DB_R134a_AT_2_Values".Status.Flag_Cycle_abort;
   END_TRANSITION
   STEP "compr. air release 1":   // S27, max time T#10S, warning time T#7S
      supervision V := ("DB_R134a_1_StepData".Values.OperationMode <> "OP_SingleStep") AND (#"compr. air release 1".U > "DB_R134a_1_StepData"."Step"[27].MonitoringTime) AND ("DB_R134a_1_StepData".Values.CycleStatus = "CS_PROCESS_RUNNING=0");
              N    "DB_R134a_1_StepData".Values.CurrentStep:= 27
          S1  R    "DB_R134a_AT_2_Values".Status.Flag_Cycle_abort
   END_STEP
   TRANSITION "AbortStep (27)" FROM "compr. air release 1" TO "compr. air release 2"   // T127, jump
      := (("DB_R134a_1_StepData".Values.CycleStatus >= "CS_USER_ABORT=2") AND ((("DB_R134a_1_StepData".Values.OperationMode = "OP_AUTOMATIC") AND ("DB_R134a_1_StepData"."Step"[27].History.ElapsedTime > "DB_R134a_1_StepData"."Step"[27].WaitingTime)) OR ("DB_R134a_1_StepData".Values.SingleStep AND ("DB_R134a_1_StepData".Values.OperationMode = "OP_SingleStep"))) AND NOT "DB_R134a_AT_2_Values".Status.Flag_Cycle_abort) OR "DB_R134a_AT_2_Values".Status.Flag_Cycle_abort;
   END_TRANSITION
   TRANSITION "NextStep (27)" FROM "compr. air release 1" TO "compr. air release 2"   // T27
      := ("DB_R134a_1_StepData".Values.CycleStatus = "CS_PROCESS_RUNNING=0") AND ((("DB_R134a_1_StepData".Values.OperationMode = "OP_AUTOMATIC") AND ("DB_R134a_1_StepData"."Step"[27].History.ElapsedTime > "DB_R134a_1_StepData"."Step"[27].WaitingTime) AND ("DB_R134a_1_StepData"."Step"[27].History.Values[5] <= "DB_R134a_1_StepData"."Step"[27].Setpoint[5])) OR ("DB_R134a_1_StepData".Values.SingleStep AND ("DB_R134a_1_StepData".Values.OperationMode = "OP_SingleStep"))) AND NOT "DB_R134a_AT_2_Values".Status.Flag_Cycle_abort;
   END_TRANSITION
   STEP "compr. air test test":   // S22, max time T#10S, warning time T#7S
      supervision V := ("DB_R134a_1_StepData".Values.OperationMode <> "OP_SingleStep") AND (#"compr. air test test".U > "DB_R134a_1_StepData"."Step"[22].MonitoringTime) AND ("DB_R134a_1_StepData".Values.CycleStatus = "CS_PROCESS_RUNNING=0");
              N    "DB_R134a_1_StepData".Values.CurrentStep:= 22
          S1  R    "DB_R134a_AT_2_Values".Status.Flag_Cycle_abort
   END_STEP
   TRANSITION "AbortStep (22)" FROM "compr. air test test" TO "compr. air release 1"   // T122, jump
      := "DB_R134a_AT_2_Values".Status.Flag_Cycle_abort;
   END_TRANSITION
   TRANSITION "NextStep (22)" FROM "compr. air test test" TO "compr. air release 1"   // T22
      := ("DB_R134a_1_StepData".Values.CycleStatus = "CS_PROCESS_RUNNING=0") AND ((("DB_R134a_1_StepData".Values.OperationMode = "OP_AUTOMATIC") AND ("DB_R134a_1_StepData"."Step"[22].History.ElapsedTime > "DB_R134a_1_StepData"."Step"[22].WaitingTime) AND ("DB_R134a_1_StepData"."Step"[22].History.Values[5] >= "DB_R134a_1_StepData"."Step"[22].Setpoint[5]) AND ("DB_R134a_1_StepData"."Step"[22].History.Values[6] >= "DB_R134a_1_StepData"."Step"[22].Setpoint[6])) OR ("DB_R134a_1_StepData".Values.SingleStep AND ("DB_R134a_1_StepData".Values.OperationMode = "OP_SingleStep"))) AND NOT "DB_R134a_AT_2_Values".Status.Flag_Cycle_abort;
   END_TRANSITION
   STEP "compr. air stabilize":   // S21, max time T#10S, warning time T#7S
      supervision V := ("DB_R134a_1_StepData".Values.OperationMode <> "OP_SingleStep") AND (#"compr. air stabilize".U > "DB_R134a_1_StepData"."Step"[21].MonitoringTime) AND ("DB_R134a_1_StepData".Values.CycleStatus = "CS_PROCESS_RUNNING=0") AND ("DB_R134a_AT_2_Values".OperationMode.SteadyCompressedAirTest = "OP_NO_SteadyComprAirTest");
              N    "DB_R134a_1_StepData".Values.CurrentStep:= 21
          S1  R    "DB_R134a_AT_2_Values".Status.Flag_Cycle_abort
   END_STEP
   TRANSITION "AbortStep (21)" FROM "compr. air stabilize" TO "compr. air release 1"   // T121, jump
      := "DB_R134a_AT_2_Values".Status.Flag_Cycle_abort;
   END_TRANSITION
   TRANSITION "NextStep (21)" FROM "compr. air stabilize" TO "compr. air test test"   // T21
      := ("DB_R134a_1_StepData".Values.CycleStatus = "CS_PROCESS_RUNNING=0") AND ((("DB_R134a_1_StepData".Values.OperationMode = "OP_AUTOMATIC") AND ("DB_R134a_1_StepData"."Step"[21].History.ElapsedTime > "DB_R134a_1_StepData"."Step"[21].WaitingTime) AND ("DB_R134a_1_StepData"."Step"[21].History.Values[5] >= "DB_R134a_1_StepData"."Step"[21].Setpoint[5]) AND ("DB_R134a_AT_2_Values".OperationMode.SteadyCompressedAirTest = "OP_NO_SteadyComprAirTest")) OR ("DB_R134a_1_StepData".Values.SingleStep AND ("DB_R134a_1_StepData".Values.OperationMode = "OP_SingleStep"))) AND NOT "DB_R134a_AT_2_Values".Status.Flag_Cycle_abort;
   END_TRANSITION
   STEP "compr.air fill":   // S20, max time T#10S, warning time T#7S
      supervision V := ("DB_R134a_1_StepData".Values.OperationMode <> "OP_SingleStep") AND (#"compr.air fill".U > "DB_R134a_1_StepData"."Step"[20].MonitoringTime) AND ("DB_R134a_1_StepData".Values.CycleStatus = "CS_PROCESS_RUNNING=0");
              N    "DB_R134a_1_StepData".Values.CurrentStep:= 20
          S1  R    "DB_R134a_AT_2_Values".Status.Flag_Cycle_abort
   END_STEP
   TRANSITION "AbortStep (20)" FROM "compr.air fill" TO "compr. air release 1"   // T120, jump
      := "DB_R134a_AT_2_Values".Status.Flag_Cycle_abort;
   END_TRANSITION
   TRANSITION "NextStep (20)" FROM "compr.air fill" TO "compr. air stabilize"   // T20
      := ("DB_R134a_1_StepData".Values.CycleStatus = "CS_PROCESS_RUNNING=0") AND ((("DB_R134a_1_StepData".Values.OperationMode = "OP_AUTOMATIC") AND ("DB_R134a_1_StepData"."Step"[20].History.ElapsedTime > "DB_R134a_1_StepData"."Step"[20].WaitingTime) AND ("DB_R134a_1_StepData"."Step"[20].History.Values[5] >= "DB_R134a_1_StepData"."Step"[20].Setpoint[5])) OR ("DB_R134a_1_StepData".Values.SingleStep AND ("DB_R134a_1_StepData".Values.OperationMode = "OP_SingleStep"))) AND NOT "DB_R134a_AT_2_Values".Status.Flag_Cycle_abort;
   END_TRANSITION
   STEP "systemtest 1 pressure":   // S16, max time T#10S, warning time T#7S
      supervision V := ("DB_R134a_1_StepData".Values.OperationMode <> "OP_SingleStep") AND (#"systemtest 1 pressure".U > "DB_R134a_1_StepData"."Step"[16].MonitoringTime) AND ("DB_R134a_1_StepData".Values.CycleStatus = "CS_PROCESS_RUNNING=0");
              N    "DB_R134a_1_StepData".Values.CurrentStep:= 16
          S1  R    "DB_R134a_AT_2_Values".Status.Flag_Cycle_abort
   END_STEP
   TRANSITION "OptionStep (16)" FROM "systemtest 1 pressure" TO "test connection to vehicle"   // T216, jump
      := ("DB_R134a_1_StepData".Values.CycleStatus = "CS_PROCESS_RUNNING=0") AND ((("DB_R134a_1_StepData".Values.OperationMode = "OP_AUTOMATIC") AND ("DB_R134a_1_StepData"."Step"[16].History.ElapsedTime > "DB_R134a_1_StepData"."Step"[16].WaitingTime) AND ("DB_R134a_1_StepData"."Step"[16].History.Values[5] < "DB_R134a_1_StepData"."Step"[16].Setpoint[5])) OR ("DB_R134a_1_StepData".Values.SingleStep AND ("DB_R134a_1_StepData".Values.OperationMode = "OP_SingleStep"))) AND ("DB_R134a_AT_2_Values".OperationMode.CompressedAirTest = "OP_BYPASS_AIRPRESSURE_TEST") AND NOT "DB_R134a_AT_2_Values".Status.Flag_Cycle_abort;
   END_TRANSITION
   TRANSITION "AbortStep (16)" FROM "systemtest 1 pressure" TO "release system"   // T116
      := "DB_R134a_AT_2_Values".Status.Flag_Cycle_abort;
   END_TRANSITION
   TRANSITION "NextStep (16)" FROM "systemtest 1 pressure" TO "compr.air fill"   // T16
      := ("DB_R134a_1_StepData".Values.CycleStatus = "CS_PROCESS_RUNNING=0") AND ((("DB_R134a_1_StepData".Values.OperationMode = "OP_AUTOMATIC") AND ("DB_R134a_1_StepData"."Step"[16].History.ElapsedTime > "DB_R134a_1_StepData"."Step"[16].WaitingTime) AND ("DB_R134a_1_StepData"."Step"[16].History.Values[5] <= "DB_R134a_1_StepData"."Step"[16].Setpoint[5])) OR ("DB_R134a_1_StepData".Values.SingleStep AND ("DB_R134a_1_StepData".Values.OperationMode = "OP_SingleStep"))) AND ("DB_R134a_AT_2_Values".OperationMode.CompressedAirTest = "OP_WITH_AIRPRESSURE_TEST") AND NOT "DB_R134a_AT_2_Values".Status.Flag_Cycle_abort;
   END_TRANSITION
   STEP "change sequence":   // S15, max time T#10S, warning time T#7S
              N    "DB_R134a_1_StepData".Values.CurrentStep:= 15
          S1  R    "DB_R134a_AT_2_Values".Status.Flag_Cycle_abort
   END_STEP
   TRANSITION "AbortStep (15)" FROM "change sequence" TO "cycle end"   // T115, jump
      := "DB_R134a_AT_2_Values".Status.Flag_Cycle_abort;
   END_TRANSITION
   TRANSITION "NextStep (15)" FROM "change sequence" TO "systemtest 1 pressure"   // T15
      := ("DB_R134a_1_StepData".Values.CycleStatus = "CS_PROCESS_RUNNING=0") AND ((("DB_R134a_1_StepData".Values.OperationMode = "OP_AUTOMATIC") AND ("DB_R134a_1_StepData"."Step"[15].History.ElapsedTime > "DB_R134a_1_StepData"."Step"[15].WaitingTime)) OR ("DB_R134a_1_StepData".Values.SingleStep AND ("DB_R134a_1_StepData".Values.OperationMode = "OP_SingleStep"))) AND NOT "DB_R134a_AT_2_Values".Status.Flag_Cycle_abort;
   END_TRANSITION
   STEP "evacuating vacuumpipe":   // S11, max time T#10S, warning time T#7S
      supervision V := ("DB_R134a_1_StepData".Values.OperationMode <> "OP_SingleStep") AND (#"evacuating vacuumpipe".U > "DB_R134a_1_StepData"."Step"[11].MonitoringTime) AND ("DB_R134a_1_StepData".Values.CycleStatus = "CS_PROCESS_RUNNING=0");
              N    "DB_R134a_1_StepData".Values.CurrentStep:= 11
          S1  R    "DB_R134a_AT_2_Values".Status.Flag_Cycle_abort
   END_STEP
   TRANSITION "AbortStep (11)" FROM "evacuating vacuumpipe" TO "cycle end"   // T111, jump
      := "DB_R134a_AT_2_Values".Status.Flag_Cycle_abort;
   END_TRANSITION
   TRANSITION "NextStep (11)" FROM "evacuating vacuumpipe" TO "change sequence"   // T11
      := ("DB_R134a_1_StepData".Values.CycleStatus = "CS_PROCESS_RUNNING=0") AND ((("DB_R134a_1_StepData".Values.OperationMode = "OP_AUTOMATIC") AND ("DB_R134a_1_StepData"."Step"[11].History.ElapsedTime > "DB_R134a_1_StepData"."Step"[11].WaitingTime) AND ("DB_R134a_1_StepData"."Step"[11].History.Values[1] <= "DB_R134a_1_StepData"."Step"[11].Setpoint[1])) OR ("DB_R134a_1_StepData".Values.SingleStep AND ("DB_R134a_1_StepData".Values.OperationMode = "OP_SingleStep"))) AND NOT "DB_R134a_AT_2_Values".Status.Flag_Cycle_abort;
   END_TRANSITION
   STEP "cycle start":   // S10, max time T#10S, warning time T#7S
              N    "DB_R134a_1_StepData".Values.CurrentStep:= 10
          S1  R    "DB_R134a_AT_2_Values".Status.Flag_Cycle_abort
   END_STEP
   TRANSITION "OptionStep (10)" FROM "cycle start" TO "change sequence"   // T210, jump: ### IBN_TRUE ### Abbruchbedingung prüfen / korrigieren
      := ("DB_R134a_1_StepData".Values.CycleStatus = "CS_PROCESS_RUNNING=0") AND ((("DB_R134a_1_StepData".Values.OperationMode = "OP_AUTOMATIC") AND ("DB_R134a_1_StepData"."Step"[10].History.ElapsedTime > "DB_R134a_1_StepData"."Step"[10].WaitingTime)) OR ("DB_R134a_1_StepData".Values.SingleStep AND ("DB_R134a_1_StepData".Values.OperationMode = "OP_SingleStep"))) AND ("DB_R134a_AT_2_Values".OperationMode.AdaptionTest = "OP_BYPASS_ADAPTIONTEST") AND NOT "DB_R134a_AT_2_Values".Status.Flag_Cycle_abort;
   END_TRANSITION
   TRANSITION "AbortStep (10)" FROM "cycle start" TO "cycle end"   // T110, jump
      := "DB_R134a_AT_2_Values".Status.Flag_Cycle_abort;
   END_TRANSITION
   TRANSITION "NextStep (10)" FROM "cycle start" TO "evacuating vacuumpipe"   // T10
      := ("DB_R134a_1_StepData".Values.CycleStatus = "CS_PROCESS_RUNNING=0") AND ((("DB_R134a_1_StepData".Values.OperationMode = "OP_AUTOMATIC") AND ("DB_R134a_1_StepData"."Step"[10].History.ElapsedTime > "DB_R134a_1_StepData"."Step"[10].WaitingTime)) OR ("DB_R134a_1_StepData".Values.SingleStep AND ("DB_R134a_1_StepData".Values.OperationMode = "OP_SingleStep"))) AND ("DB_R134a_AT_2_Values".OperationMode.AdaptionTest = "OP_WITH_ADAPTIONTEST") AND NOT "DB_R134a_AT_2_Values".Status.Flag_Cycle_abort;
   END_TRANSITION
   STEP "venting adapter":   // S4, max time T#10S, warning time T#7S
              N    "DB_R134a_1_StepData".Values.CurrentStep:= 4
          S1  R    "DB_R134a_AT_2_Values".Status.Flag_Cycle_abort
   END_STEP
   TRANSITION "NextStep (4)" FROM "venting adapter" TO "cycle start"   // T4
      := NOT "DB_R134a_AT_2_Values".Status.AdapterHomePosHP AND NOT "DB_R134a_AT_2_Values".Status.AdapterHomePosLP AND "DB_R134a_AT_2_Values".Status.CycleStartReady AND "DB_R134a_AT_2_Values".Status.CycleStartStop;
   END_TRANSITION
   TRANSITION "OptionStep (2)" FROM "venting adapter" TO "stand by"   // T2, jump
      := ("DB_R134a_AT_2_Values".Status.AdapterHomePosHP AND "DB_R134a_AT_2_Values".Status.AdapterHomePosLP) OR NOT "DB_R134a_BU_Values".Module.On;
   END_TRANSITION
   INITIAL_STEP "stand by":   // S1, max time T#10S, warning time T#7S
              N    "DB_R134a_1_StepData".Values.CurrentStep:= 0
          S1  R    "DB_R134a_AT_2_Values".Status.Flag_Cycle_abort
   END_STEP
   TRANSITION "NextStep (1)" FROM "stand by" TO "venting adapter"   // T1
      := (NOT "DB_R134a_AT_2_Values".Status.AdapterHomePosHP OR NOT "DB_R134a_AT_2_Values".Status.AdapterHomePosLP) AND "DB_R134a_BU_Values".Module.On;
   END_TRANSITION
   STEP "filling 1 PAG oil":   // S36, max time T#10S, warning time T#7S
      supervision V := ("DB_R134a_1_StepData".Values.OperationMode <> "OP_SingleStep") AND (#"filling 1 PAG oil".U > "DB_R134a_1_StepData"."Step"[36].MonitoringTime) AND ("DB_R134a_1_StepData".Values.CycleStatus = "CS_PROCESS_RUNNING=0");
              N    "DB_R134a_1_StepData".Values.CurrentStep:= 36
          S1  R    "DB_R134a_AT_2_Values".Status.Flag_Cycle_abort
   END_STEP
   TRANSITION "NextStep (36)" FROM "filling 1 PAG oil" TO "change sequence f1/f2"   // T36
      := ("DB_R134a_1_StepData".Values.CycleStatus = "CS_PROCESS_RUNNING=0") AND ((("DB_R134a_1_StepData".Values.OperationMode = "OP_AUTOMATIC") AND ("DB_R134a_1_StepData"."Step"[36].History.ElapsedTime > "DB_R134a_1_StepData"."Step"[36].WaitingTime) AND "DB_R134a_BU_Values".FlowmeterPAG.Output.VolumeDone) OR ("DB_R134a_1_StepData".Values.SingleStep AND ("DB_R134a_1_StepData".Values.OperationMode = "OP_SingleStep"))) AND NOT "DB_R134a_AT_2_Values".Status.Flag_Cycle_abort;
   END_TRANSITION
   TRANSITION "AbortStep (36)" FROM "filling 1 PAG oil" TO "release system"   // T136, jump
      := "DB_R134a_AT_2_Values".Status.Flag_Cycle_abort;
   END_TRANSITION
   STEP "change sequence f1/f2":   // S37, max time T#10S, warning time T#7S
              N    "DB_R134a_1_StepData".Values.CurrentStep:= 37
          S1  R    "DB_R134a_AT_2_Values".Status.Flag_Cycle_abort
   END_STEP
   TRANSITION "NextStep (37)" FROM "change sequence f1/f2" TO "filling 2 R134a"   // T37
      := ("DB_R134a_1_StepData".Values.CycleStatus = "CS_PROCESS_RUNNING=0") AND ((("DB_R134a_1_StepData".Values.OperationMode = "OP_AUTOMATIC") AND ("DB_R134a_1_StepData"."Step"[37].History.ElapsedTime > "DB_R134a_1_StepData"."Step"[37].WaitingTime)) OR ("DB_R134a_1_StepData".Values.SingleStep AND ("DB_R134a_1_StepData".Values.OperationMode = "OP_SingleStep"))) AND ("DB_R134a_AT_2_Values".OperationMode.Filling = "OP_WITH_FILLING") AND NOT "DB_R134a_AT_2_Values".Status.Flag_Cycle_abort;
   END_TRANSITION
   TRANSITION "AbortStep (37)" FROM "change sequence f1/f2" TO "release system"   // T137, jump
      := "DB_R134a_AT_2_Values".Status.Flag_Cycle_abort;
   END_TRANSITION
   TRANSITION "OptionStep (37)" FROM "change sequence f1/f2" TO "cycle end"   // T237, jump
      := ("DB_R134a_1_StepData".Values.CycleStatus = "CS_PROCESS_RUNNING=0") AND ((("DB_R134a_1_StepData".Values.OperationMode = "OP_AUTOMATIC") AND ("DB_R134a_1_StepData"."Step"[37].History.ElapsedTime > "DB_R134a_1_StepData"."Step"[37].WaitingTime)) OR ("DB_R134a_1_StepData".Values.SingleStep AND ("DB_R134a_1_StepData".Values.OperationMode = "OP_SingleStep"))) AND ("DB_R134a_AT_2_Values".OperationMode.Filling = "OP_BYPASS_FILLING") AND NOT "DB_R134a_AT_2_Values".Status.Flag_Cycle_abort;
   END_TRANSITION
END_FUNCTION_BLOCK
